FUNCTION_BLOCK FB_MeanFilters
VAR 
	m_windowSize : INT:= MAX_WINDOW_SIZE;
	m_buffer: ARRAY[0..MAX_WINDOW_SIZE-1] OF REAL;
	m_tail : INT;      
    m_count: INT := 0; 
	m_sum : LREAL :=0;
END_VAR
VAR CONSTANT
    MAX_WINDOW_SIZE: INT := 1000;  
END_VAR

METHOD init : BOOL
VAR_INPUT
	windowSize : INT:= MAX_WINDOW_SIZE;
END_VAR
m_windowSize := LIMIT(10, windowSize, MAX_WINDOW_SIZE);
m_sum := 0;
m_count := 0;
m_tail := 0;
END_METHOD

METHOD run : LREAL
VAR_INPUT
    newValue: REAL;        
END_VAR
IF m_count <= m_windowSize THEN
	m_count := m_count + 1;
	m_sum := (m_sum + newValue);
ELSE
	m_sum := m_sum - m_buffer[m_tail] + newValue;
END_IF
run := m_sum / m_windowSize;
m_buffer[m_tail] := newValue;
m_tail := (m_tail + 1) MOD m_windowSize;
END_METHOD

END_FUNCTION_BLOCK

(* stored: Version 1.1.0.1, ProductVersion 3.1.4024.11
   POU FB_MeanFilters: Id {a0402b55-69aa-4a05-ba1a-36b4bb51a055}, SpecialFunc None
   Method init: Id {1df21118-f241-421e-a6c7-9da0bacbe212}
   Method run: Id {5b5dcfd1-d55c-46ed-8825-10c09ee74e40} *)
